FUNCTION_BLOCK FB_ClearEventLog
VAR_INPUT
    bTrigger    : BOOL;
END_VAR
VAR_OUTPUT
    bBusy       : BOOL;
    bDone       : BOOL;
END_VAR
VAR
    fbLogger        : FB_TcEventLogger;
    bTriggerLast    : BOOL;
END_VAR

// Rising edge detection
IF bTrigger AND NOT bTriggerLast AND NOT bBusy THEN
    bBusy := TRUE;
    bDone := FALSE;
END_IF
bTriggerLast := bTrigger;

// Async clear logic
IF bBusy THEN
    IF NOT fbLogger.ClearLoggedEvents(0) THEN
        bBusy := FALSE;
        bDone := TRUE;
    END_IF
END_IF

END_FUNCTION_BLOCK

(* stored: Version 1.1.0.1, ProductVersion 3.1.4024.14
   POU FB_ClearEventLog: Id {01c317a4-3bdc-4058-a8dc-ac1b50e9e4f6}, SpecialFunc None *)
